% RSLogix 500 project I2P HANDS-ON 3 - TYLER.RSS, saved by version 10.00.00.00 %
PROJECT "UNTITLED"    % processor: Bul.1763 MicroLogix 1100 Series B %

PROGRAM FILES
  LAD 2   10 rungs

DATA FILES
  O0 OUTPUT  4 elements
  I1 INPUT  6 elements
  S2 STATUS  66 elements
  B3 BINARY  1 elements
  T4 TIMER  1 elements
  C5 COUNTER  1 elements
  R6 CONTROL  1 elements
  N7 INTEGER  1 elements
  F8 FLOAT  1 elements

LADDER 2
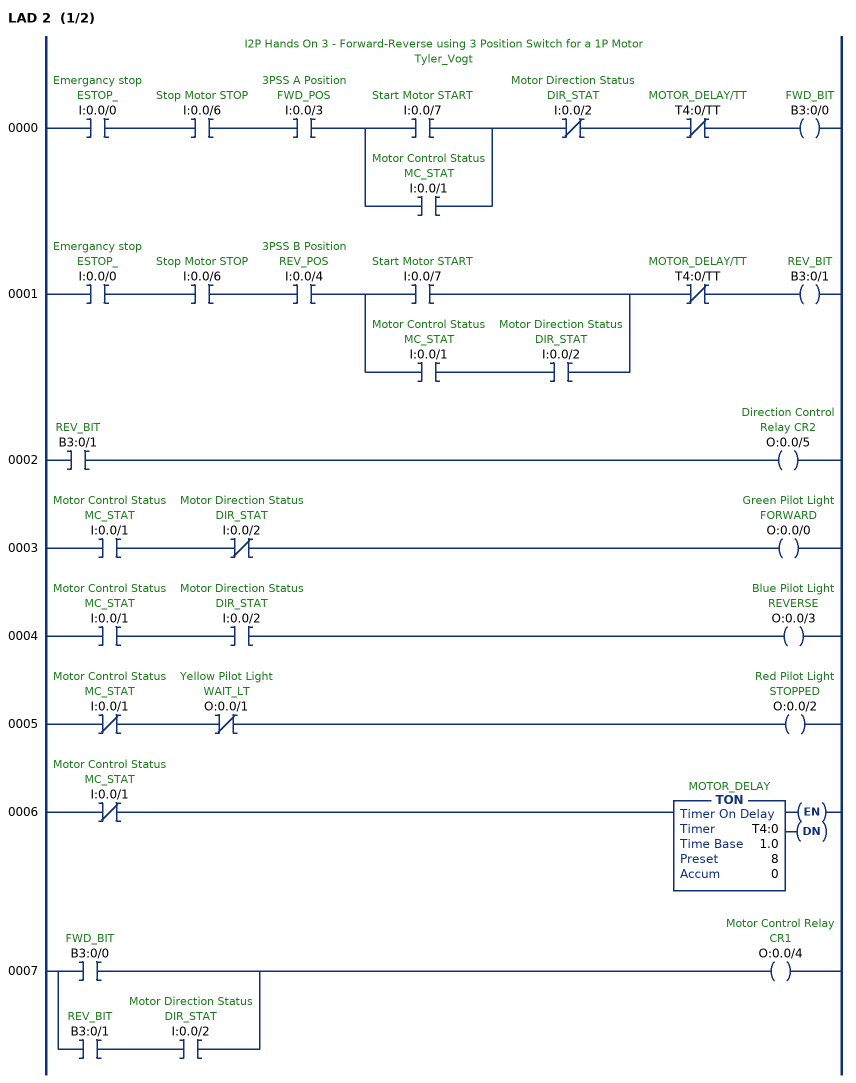
% Rung: 0 %
% I2P Hands On 3 - Forward-Reverse using 3 Position Switch for a 1P Motor
% Tyler_Vogt %
SOR XIC I:0.0/0 XIC I:0.0/6 XIC I:0.0/3 BST XIC I:0.0/7 NXB XIC I:0.0/1 BND XIO I:0.0/2 XIO T4:0/TT OTE B3:0/0 EOR
%   I:0.0/0  ESTOP_  "Emergancy stop" %
%   I:0.0/6  STOP  "Stop Motor" %
%   I:0.0/3  FWD_POS  "3PSS A Position" %
%   I:0.0/7  START  "Start Motor" %
%   I:0.0/1  MC_STAT  "Motor Control Status" %
%   I:0.0/2  DIR_STAT  "Motor Direction Status" %
%   T4:0  MOTOR_DELAY %
%   B3:0/0  FWD_BIT %
% Rung: 1 %
SOR XIC I:0.0/0 XIC I:0.0/6 XIC I:0.0/4 BST XIC I:0.0/7 NXB XIC I:0.0/1 XIC I:0.0/2 BND XIO T4:0/TT OTE B3:0/1 EOR
%   I:0.0/0  ESTOP_  "Emergancy stop" %
%   I:0.0/6  STOP  "Stop Motor" %
%   I:0.0/4  REV_POS  "3PSS B Position" %
%   I:0.0/7  START  "Start Motor" %
%   I:0.0/1  MC_STAT  "Motor Control Status" %
%   I:0.0/2  DIR_STAT  "Motor Direction Status" %
%   T4:0  MOTOR_DELAY %
%   B3:0/1  REV_BIT %
% Rung: 2 %
SOR XIC B3:0/1 OTE O:0.0/5 EOR
%   B3:0/1  REV_BIT %
%   O:0.0/5  CR2  "Direction Control Relay" %
% Rung: 3 %
SOR XIC I:0.0/1 XIO I:0.0/2 OTE O:0.0/0 EOR
%   I:0.0/1  MC_STAT  "Motor Control Status" %
%   I:0.0/2  DIR_STAT  "Motor Direction Status" %
%   O:0.0/0  FORWARD  "Green Pilot Light" %
% Rung: 4 %
SOR XIC I:0.0/1 XIC I:0.0/2 OTE O:0.0/3 EOR
%   I:0.0/1  MC_STAT  "Motor Control Status" %
%   I:0.0/2  DIR_STAT  "Motor Direction Status" %
%   O:0.0/3  REVERSE  "Blue Pilot Light" %
% Rung: 5 %
SOR XIO I:0.0/1 XIO O:0.0/1 OTE O:0.0/2 EOR
%   I:0.0/1  MC_STAT  "Motor Control Status" %
%   O:0.0/1  WAIT_LT  "Yellow Pilot Light" %
%   O:0.0/2  STOPPED  "Red Pilot Light" %
% Rung: 6 %
SOR XIO I:0.0/1 TON T4:0 1.0 8 0 EOR
%   I:0.0/1  MC_STAT  "Motor Control Status" %
%   T4:0  MOTOR_DELAY %
% Rung: 7 %
SOR BST XIC B3:0/0 NXB XIC B3:0/1 XIC I:0.0/2 BND OTE O:0.0/4 EOR
%   B3:0/0  FWD_BIT %
%   B3:0/1  REV_BIT %
%   I:0.0/2  DIR_STAT  "Motor Direction Status" %
%   O:0.0/4  CR1  "Motor Control Relay" %

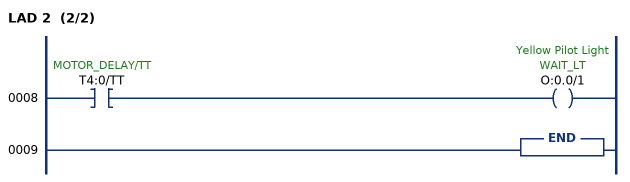
% Rung: 8 %
SOR XIC T4:0/TT OTE O:0.0/1 EOR
%   T4:0  MOTOR_DELAY %
%   O:0.0/1  WAIT_LT  "Yellow Pilot Light" %
% Rung: 9 %
SOR END EOR

DATA TABLE (non-zero values as saved)
DATA T4
% .PRE .ACC %
% T4:0 % 8 0
